TYPE C13336MppcConfig EXTENDS DeviceConfiguration :
STRUCT
	SerialCommunication : SerialCommunication;
END_STRUCT
END_TYPE

(* stored: Version 1.1.0.1, ProductVersion 3.1.4024.4
   DUT C13336MppcConfig: Id {40089f3f-1572-47ce-88e7-25f6f09826bf} *)
